FUNCTION_BLOCK SM_TransferLine EXTENDS StateMachine
VAR_INPUT
END_VAR
VAR_OUTPUT
END_VAR
VAR
	
	aRollerConveyors : ARRAY[1..3] OF RollerConveyor;
	
	
	fbPalletizer : SM_Palletizer;
	fbStepWorkerReady : FB_StepWorker;
	fbStepWorkerBusy : FB_StepWorker;
	
	fbChainController : FB_ChainController;
	
	scBeltConveyors : 
		SC_BeltConveyors := 
		(
			init_uiChainNumber := 1, 
			init_sChainName  := 'scBeltConveyors',
			init_rChainController := fbChainController
		);
		
	scPostPalletizer : 
		SC_PostPalletizer := 
		(
			init_uiChainNumber := 2, 
			init_sChainName  := 'scPostPalletizer',
			init_rChainController := fbChainController
		);
		
	scPrePalletizer : 
		SC_PrePalletizer := 
		(
			init_uiChainNumber := 3, 
			init_sChainName  := 'scPrePalletizer',
			init_rChainController := fbChainController
		);
 
	fbTrig : R_TRIG;
	uiPackageCounter : UINT;
	i : UINT;
	bPackageOnTheWay : BOOL;
END_VAR

SUPER^();
fbPalletizer();
scBeltConveyors(ioPalletizer := fbPalletizer);

METHOD PROTECTED Busy : BOOL
VAR_INPUT
END_VAR
CASE fbStepWorkerBusy.uiStep OF

END_CASE
END_METHOD

METHOD PROTECTED  Error : BOOL
VAR_INPUT
END_VAR
END_METHOD

METHOD PROTECTED  Idle : BOOL
VAR_INPUT
END_VAR
END_METHOD

METHOD PROTECTED  Init : BOOL
VAR_INPUT
END_VAR
Start();
END_METHOD

METHOD PROTECTED  Prepare : BOOL
VAR_INPUT
END_VAR
END_METHOD

METHOD PROTECTED  Ready : BOOL
VAR_INPUT
END_VAR
END_METHOD

METHOD PROTECTED  Waiting : BOOL
VAR_INPUT
END_VAR
END_METHOD

END_FUNCTION_BLOCK

(* stored: Version 1.1.0.1, ProductVersion 3.1.4024.2
   POU SM_TransferLine: Id {2e7b366f-b9ef-4b13-bd70-7031bb32b800}, SpecialFunc None
   Method Busy: Id {3dde4417-0d0c-49da-9bd9-97065e9ed964}
   Method Error: Id {dcf9a9b3-729d-4763-8c13-3d1ffd1dfd1e}
   Method Idle: Id {93f70726-6e20-4944-9007-789a6a898f24}
   Method Init: Id {4357aa31-540d-408d-bbfa-5ee1874096be}
   Method Prepare: Id {702c85df-2da8-4392-a504-15b946826c27}
   Method Ready: Id {4f0f5542-23e8-48a2-84b3-069ccd15f633}
   Method Waiting: Id {8f7a7b39-5942-438f-a1c3-fcbbad8d2ba6} *)
